// Injects a previously persisted value into an otherwise fresh instance.
// This tests startup policy, NOT actual TwinCAT persistent-image durability.
FUNCTION_BLOCK FB_AnalogOutputRestart_Probe EXTENDS TcForge.FB_AnalogOutput
VAR_INPUT
    simulatedBootDataLoaded : BOOL := TRUE;
    simulatedOldBootData : BOOL;
END_VAR

SUPER^();

METHOD PUBLIC SeedSavedCommand
VAR_INPUT
    value : REAL;
END_VAR
_savedCommand := value;
_savedCommandValid := TRUE;
END_METHOD

// Policy probe: reset volatile arming only; not a runtime/persistent-image test.
METHOD PUBLIC SimulateStartup
_startup := TRUE;
_commandReceived := FALSE;
_armed := FALSE;
_forceSafe := FALSE;
_safeRequested := FALSE;
_requestSync := 0.0;
END_METHOD

METHOD PROTECTED _HasTrustedPersistentImage : BOOL
// Local probe inputs only: never mutate TwinCAT system information.
_HasTrustedPersistentImage := simulatedBootDataLoaded AND NOT simulatedOldBootData;
END_METHOD

END_FUNCTION_BLOCK

(* stored: Version 1.1.0.1
   POU FB_AnalogOutputRestart_Probe: Id {ebbca1f8-d594-4e16-8e01-6a69b7b6ee85}
   Method SeedSavedCommand: Id {61a14c7d-e2c0-43a8-b919-62c5c8be93eb}
   Method SimulateStartup: Id {578ac2f4-3463-4339-80c5-977d64b8c14b}
   Method _HasTrustedPersistentImage: Id {ad6e76eb-ef94-4632-b781-d0d349f32271} *)
